# EPICS IOC start-up script: require/3.1.2/siteMods/mrfioc2/2.2.1rc3/evr.iocsh
#!
mrmEvrSetupPCI "$(OBJ=EVR)" "$(PCIID)"

dbLoadRecords "$(FILE_DB=evr-mtca-300u-ess.db)" "P=$(P), OBJ=$(OBJ=EVR), FEVT=$(TS_CLK=88.0525)"

# needed with software timestamp [ns] source w/o RT thread scheduling
var evrMrmTimeNSOverflowThreshold 500000000
